RoboDK station: Bachelorarbeit.rdk

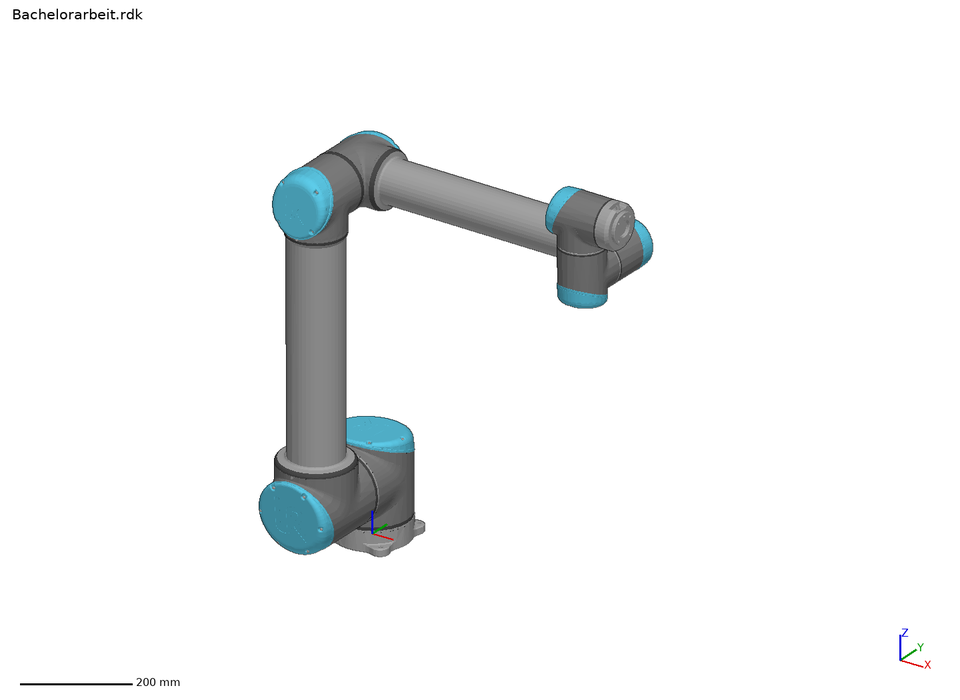
[picture v0: the station drawn from its stored meshes, robots at their saved joint values, targets as dots, program paths as lines]
Station Bachelorarbeit (saved by RoboDK 5.6.7). Poses are relative to the parent item; angles as X-Y-Z fixed-axis rotations.
Station parameters (name, value as stored): LIN64
  - frame UR10 Base at (0, 0, 0) mm
    - robot UR10: 6 axes, payload 10 kg, reach 1300 mm, repeatability 0.1 mm, weight 28.9 kg
        modified DH rows (alpha deg, a mm, theta deg, d mm): 0, 0, 0, 128; 90, 0, 180, 0; 0, 612.7, 0, 0; 0, 571.6, 0, 163.9; -90, 0, 0, 115.7; 90, 0, 180, 92.2
        joint limits [-360, -360, -360, -360, -360, -360] to [360, 360, 360, 360, 360, 360]; home [0, -90, -90, 0, 90, 0]; saved at [0, -90, -90, 0, 90, 0]
  - Python program Prog1 (listed below)

--- Python program Prog1 ---
# Import RoboDK API python libraries
from robodk.robolink import *
from robodk.robomath import *
# Import RTDE python libraries
from rtde_control import RTDEControlInterface as RTDEControl
from rtde_receive import RTDEReceiveInterface as RTDEReceive
# Import data display python libraries
import pandas as pd
import matplotlib.pyplot as plt
# Import other python libraries
import datetime
import math
import os
import psutil
import sys

# Link to RoboDK
RDK = Robolink()

# Program example:
robot = RDK.ItemUserPick('Select a robot', ITEM_TYPE_ROBOT)
if not robot.Valid():
    raise Exception('No robot selected or available')

# get the current position of the TCP with respect to the reference frame:
# (4x4 matrix representing position and orientation)
target_ref = robot.Pose()
pos_ref = target_ref.Pos()
print("Drawing a polygon around the target: ")
print(Pose_2_TxyzRxyz(target_ref))

# move the robot to the first point:
robot.MoveJ(target_ref)

# It is important to provide the reference frame and the tool frames when generating programs offline
robot.setPoseFrame(robot.PoseFrame())
robot.setPoseTool(robot.PoseTool())
robot.setRounding(10)  # Set the rounding parameter (Also known as: CNT, APO/C_DIS, ZoneData, Blending radius, cornering, ...)
robot.setSpeed(200)  # Set linear speed in mm/s

# Set the number of sides of the polygon:
n_sides = 6
R = 100

# make a hexagon around reference target:
for i in range(n_sides + 1):
    ang = i * 2 * pi / n_sides  #angle: 0, 60, 120, ...

    #-----------------------------
    # Movement relative to the reference frame
    # Create a copy of the target
    target_i = Mat(target_ref)
    pos_i = target_i.Pos()
    pos_i[0] = pos_i[0] + R * cos(ang)
    pos_i[1] = pos_i[1] + R * sin(ang)
    target_i.setPos(pos_i)
    print("Moving to target %i: angle %.1f" % (i, ang * 180 / pi))
    print(str(Pose_2_TxyzRxyz(target_i)))
    robot.MoveL(target_i)
    print("/n")
    print(robot.Pose())
    print(robot.Pose().Pos())
    print("/n")

    #-----------------------------
    # Post multiply: relative to the tool
    #target_i = target_ref * rotz(ang) * transl(R,0,0) * rotz(-ang)
    #robot.MoveL(target_i)

# move back to the center, then home:
robot.MoveL(target_ref)

print('Done')


# Add other program
import plot_test
#import getData
